TYPE SafetyHydraulicsAndSafetyIOStatuses :
STRUCT
	///Is the I/O in a healthy state?
	healthStatus: HealthStatus;
END_STRUCT
END_TYPE

(* stored: Version 1.1.0.1, ProductVersion 3.1.4019.2
   DUT SafetyHydraulicsAndSafetyIOStatuses: Id {fd08ed41-0f35-46e6-9b33-dc08044f7ba0} *)
